PROGRAM MAIN
VAR
	Error			: BOOL;
	SystemReboot	: NT_REBOOT;
	Reboot			: BOOL;
	MsgUpdateTimer	: TON;
	MsgUpdatePeriod	: TIME := T#50MS;
	TimerResetDelay	: INT := 25;
	TimerResetCounter	: INT;
	Version			: REAL := 1.0;
	
	State			: (DEFAULT, INIT, IDLE, RUN, ERROR);
	PrevState		: (DEFAULT, INIT, IDLE, RUN, ERROR);
	StateEntry 		: BOOL;
END_VAR

Harv.ReadHw();

MsgUpdateTimer.PT := MsgUpdatePeriod;

IF PrevState <> State THEN
	StateEntry := TRUE;
	PrevState := State;
ELSE
	StateEntry := FALSE;
END_IF

CASE State OF
	DEFAULT:
		//
	INIT:
		//
	IDLE:
		//
	RUN:
		//
	ERROR:
		//
END_CASE

//IF Error THEN
//	HARV.ErrorLog.AddMsg(TimeStamp := Harv.TimeTracker.TimeStamp, Location := 'MAIN', ErrorCode := 1234, Description := 'TEST');
//	Error := FALSE;
//END_IF

IF MsgUpdateTimer.Q THEN
	TimerResetCounter := TimerResetCounter + 1;
	IF TimerResetCounter = TimerResetDelay THEN
		TimerResetCounter := 0;
		MsgUpdateTimer.IN := FALSE;
	END_IF
ELSE
	TimerResetCounter := 0;
	MsgUpdateTimer.IN := TRUE;
END_IF

SystemReboot(NETID := '', START := Reboot);

MsgUpdateTimer();
Harv.TimeTracker();
Harv.DriveSys();
Harv.TiltControl();
Harv.WriteHw();

END_PROGRAM

(* stored: Version 1.1.0.1, ProductVersion 3.1.4024.15
   POU MAIN: Id {3586711d-1897-42d6-afda-493964a09e79}, SpecialFunc None *)
